FUNCTION Convert_UINT_TO_ULINT : Hresult
VAR_INPUT
	in : UINT;
	out : REFERENCE TO ULINT;
END_VAR
VAR
	converted : ULINT;
END_VAR

converted := UINT_TO_ULINT(in);

IF (ULINT_TO_UINT(converted) <> in) THEN
	Convert_UINT_TO_ULINT := INCOMPATIBLE;
	RETURN;
END_IF

out := converted;

END_FUNCTION

(* stored: Version 1.1.0.1, ProductVersion 3.1.4024.12
   POU Convert_UINT_TO_ULINT: Id {05e1e746-5a69-49a8-aeb9-e137e506c509}, SpecialFunc None *)
